{attribute 'call_after_init'}
FUNCTION_BLOCK FB_CreateTwoTestsWithSameName EXTENDS TcUnit.FB_TestSuite IMPLEMENTS TcUnit.I_RunnableTestSuite
VAR
    Assert : TcUnit.FB_Assert;
END_VAR

METHOD FB_init : BOOL
VAR_INPUT
	bInitRetains : BOOL; // if TRUE, the retain variables are initialized (warm start / cold start)
	bInCopyCode : BOOL;  // if TRUE, the instance afterwards gets moved into the copy code (online change)
END_VAR
SUPER^.RegisterTestSuite(THIS^);
END_METHOD

METHOD RunTests : TCUNIT.E_TestSuiteRunState
TestOne();
TestOne_Again();

RunTests := TCUNIT.E_TestSuiteRunState.FINISHED;
END_METHOD

METHOD PRIVATE TestOne
VAR
    a : INT := 55;
    b : INT := 55;
END_VAR
TEST('TestOne');

Assert.AssertEquals_INT(Expected := a,
                        Actual := b,
                        Message := 'A does not equal B');
END_METHOD

METHOD PRIVATE TestOne_Again
VAR
    a : INT := 55;
    b : INT := 55;
END_VAR
TEST('TestOne');

Assert.AssertEquals_INT(Expected := a,
                        Actual := b,
                        Message := 'A does not equal B again');
END_METHOD

END_FUNCTION_BLOCK

(* stored: Version 1.1.0.1, ProductVersion 3.1.4022.12
   POU FB_CreateTwoTestsWithSameName: Id {7b1f39ab-8960-43b8-8ec6-8f13e574f736}, SpecialFunc None
   Method FB_init: Id {10367bbb-5caa-4524-936d-517e6525e89c}
   Method RunTests: Id {77d08c3d-574c-4b3d-8da4-13a3c806b4ed}
   Method TestOne: Id {a0db3538-83d9-431d-9b73-12250812435f}
   Method TestOne_Again: Id {01798474-e702-41c3-94c8-ec7fd2bc4723} *)
